PROGRAM Transporteren_order
VAR
	currentState : Taks_2 : Task_2.Inladen;
	
END_VAR

CASE currentState OF
	Task_2.Inladen:
	//Inladen van de order die is verwerkt in taak 1
	IF 
END_CASE

END_PROGRAM

(* stored: Version 1.1.0.1, ProductVersion 3.1.4024.12
   POU Transporteren_order: Id {cf28c6dd-7fed-4d27-8b70-7f0672827bc6}, SpecialFunc None *)
